{attribute 'qualified_only'}
{attribute 'global_init_slot' := '40000'}
VAR_GLOBAL
	Param_PickPlace: stParam_PickPlace;
	Param_Counter: stParam_Counter;

END_VAR

(* stored: Version 1.1.0.1, ProductVersion 3.1.4026.18
   GVL LIBRARY: Id {81dfd880-4bdc-475a-8ac4-f0bc27508dae} *)
